(* IEC 61131-3 sources: OMJSON/, 3 files *)

(* ---- OMJSON.typ ---- *)
(********************************************************************
 * COPYRIGHT --
 ********************************************************************
 * Library: OMJSON
 * File: OMJSON.typ
 * Author: davidblackburn
 * Created: September 22, 2014
 ********************************************************************
 * Data types of library OMJSON
 ********************************************************************)

TYPE
	JSON_WS_OPCODE_enum :
		(
		JSON_WS_OPCODE_CONTINUATION := 0, (*Not supported*)
		JSON_WS_OPCODE_TEXT := 1,
		JSON_WS_OPCODE_BINARY := 2, (*Not supported*)
		JSON_WS_OPCODE_CLOSE := 8,
		JSON_WS_OPCODE_PING := 9, (*Not supported*)
		JSON_WS_OPCODE_PONG := 10 (*Not supported*)
		);
	JSON_ERR_enum :
		(
		JSON_ERR_INVALIDINPUT := 50000,
		JSON_ERR_MEMALLOC,
		JSON_ERR_MAXLEVELREACHED,
		JSON_ERR_PARSE,
		JSON_ERR_HUH,
		JSON_ERR_CACHEFULLITEMS,
		JSON_ERR_CACHEFULLVARS,
		JSON_ERR_CACHEEMPTY,
		JSON_ERR_MAXITERATIONS,
		JSON_ERR_WS_KEYNOTFOUND,
		JSON_ERR_WS_FRAGMENT,
		JSON_ERR_WS_RSV,
		JSON_ERR_WS_OPCODE,
		JSON_ERR_WS_MASK,
		JSON_ERR_WS_PAYLOADLENGTH,
		JSON_ERR_TCP_FRAGMENT,
		JSON_ERR_TCP_BAD_PACKET,
		JSON_ERR_NO_LICENSE,
		JSON_ERR_WS_MAX_CLIENTS,
		JSON_ERR_WS_INVALID_MAX_CLIENTS,
		JSON_ERR_WS_,
		JSON_ERR_
		);
	jsonWSS_client_info_typ : 	STRUCT
		Connected : BOOL;
		TimeSinceLastRequest_ms : UDINT;
		ClientIP : STRING[TCPCOMM_STRLEN_IPADDRESS];
		ClientPort : UINT;
	END_STRUCT;
	jsonWSS_client_debug_typ : 	STRUCT
		socketConnectCount : DINT;
		websocketConnectCount : DINT;
		socketDisconnectCountTimeout : DINT;
		socketDisconnectCountOpcode : DINT;
		socketDisconnectCountError : DINT;
		socketDisconnectCountRecvLength0 : DINT;
		socketInvalidCountError : DINT;
		noDataCount : DINT;
		dataCount : DINT;
		justRightCount : DINT;
		tooBigCount : DINT;
		tooSmallCount : DINT;
		doubleDataCount : DINT;
		oldDataReceived : BOOL;
	END_STRUCT;
	jsonWSServer_int_client_typ : 	STRUCT
		tcpStream : TCPStream_typ;
		pReceiveData : UDINT;
		pSendData : UDINT;
		messageBuffer : datbufBuffer_typ;
		wsConnect : jsonWSConnect;
		wsConnected : BOOL;
		wsDecode : jsonWSDecode;
		wsEncode : jsonWSEncode;
		writeVariable : jsonWriteVariable;
		readVariableList : jsonReadVariableList;
		debug : jsonWSS_client_debug_typ;
		excessDataLength : DINT;
		requestTimer : TON_10ms;
		pCache : REFERENCE TO jsonCache_typ;
	END_STRUCT;
	jsonWSServer_Internal_typ : 	STRUCT
		initialized : BOOL;
		tcpServer : TCPConnectionMgr_typ;
		client : ARRAY[0..JSON_MAI_CLIENTS]OF jsonWSServer_int_client_typ;
		requestTimer : TON_10ms;
		iClient : UINT;
		connectedClients : UINT;
		maxClients : UINT;
	END_STRUCT;
	jsonHTTPServer_Int_Debug_typ : 	STRUCT
		readSendCommand : BOOL;
	END_STRUCT;
	jsonHTTPServer_Int_Write_typ : 	STRUCT
		webService : httpService;
		pUri : UDINT;
		pRequestData : UDINT;
		ResponseHeader : httpResponseHeader_t;
		processed : BOOL;
		writeVariable : jsonWriteVariable;
	END_STRUCT;
	jsonHTTPServer_Int_Read_typ : 	STRUCT
		webService : httpService;
		pUri : UDINT;
		pRequestData : UDINT;
		ResponseHeader : httpResponseHeader_t;
		processed : BOOL;
		readVariableList : jsonReadVariableList;
	END_STRUCT;
	jsonHTTPServer_Internal_typ : 	STRUCT
		initialized : BOOL;
		read : jsonHTTPServer_Int_Read_typ;
		write : jsonHTTPServer_Int_Write_typ;
		debug : jsonHTTPServer_Int_Debug_typ;
	END_STRUCT;
	jsonWSConnect_Internal_typ : 	STRUCT
		encodeBase64 : httpEncodeBase64;
	END_STRUCT;
	JSON_TYPE_enum :
		(
		JSON_TYPE_INVALID := 0,
		JSON_TYPE_OBJECT_ELEMENT,
		JSON_TYPE_ARRAY_ELEMENT
		);
	jsonStructLevel_typ : 	STRUCT
		variable : varVariable_typ;
		iItem : UINT;
		jsonType : JSON_TYPE_enum;
	END_STRUCT;
	jsonWriteVariable_Int_typ : 	STRUCT
		initialized : BOOL;
		pJSONObject : UDINT;
		pChar : UDINT;
		iStructLevel : INT;
		structLevel : ARRAY[0..JSON_MAI_STRUCTLEVEL]OF jsonStructLevel_typ;
	END_STRUCT;
	jsonReadVariableList_Int_typ : 	STRUCT
		initialized : BOOL;
		outputBuffer : datbufBuffer_typ;
		readVariable : jsonReadVariable;
	END_STRUCT;
	jsonReadVariable_Int_typ : 	STRUCT
		initialized : BOOL;
		outputBuffer : datbufBuffer_typ;
		variableName : STRING[VAR_STRLEN_NAME];
		addVariableToCache : jsonAddVariableToCache;
	END_STRUCT;
	jsonAddVariableToCache_Int_typ : 	STRUCT
		initialized : BOOL;
		iStructLevel : INT;
		structLevel : ARRAY[0..JSON_MAI_STRUCTLEVEL]OF jsonStructLevel_typ;
	END_STRUCT;
	jsonCache_typ : 	STRUCT
		iVariable : UINT;
		variable : ARRAY[0..JSON_MAI_CACHEVAR]OF jsonCacheVariable_typ;
		iItem : UINT;
		item : ARRAY[0..JSON_MAI_CACHEITEM]OF jsonCacheItem_typ;
	END_STRUCT;
	jsonCacheVariable_typ : 	STRUCT
		name : STRING[VAR_STRLEN_NAME];
		iStart : UINT;
		iEnd : UINT;
	END_STRUCT;
	jsonCacheItem_typ : 	STRUCT
		prefix : STRING[JSON_STRLEN_PREFIX];
		variable : varVariable_typ;
		suffix : STRING[JSON_STRLEN_SUFFIX];
	END_STRUCT;
	jsonReadVarNoCache_Int_typ : 	STRUCT
		initialized : BOOL;
		outputBuffer : datbufBuffer_typ;
		iStructLevel : INT;
		structLevel : ARRAY[0..JSON_MAI_STRUCTLEVEL]OF jsonStructLevel_typ;
	END_STRUCT;
END_TYPE

(* ---- OMJSON.fun ---- *)
(********************************************************************
 * COPYRIGHT --
 ********************************************************************
 * Library: OMJSON
 * File: OMJSON.fun
 * Author: davidblackburn
 * Created: September 22, 2014
 ********************************************************************
 * Functions and function blocks of library OMJSON
 ********************************************************************)

FUNCTION_BLOCK jsonWebSocketServer (*Serve variables via JSON and WebSockets*) (*$GROUP=User*)
	VAR_INPUT
		pCacheArray : UDINT; (*Address of the variable cache array. Number of elements in array needs to be equal to numClients*)
		maxClients : UINT; (*Number of clients supported at a time. 0 defaults to 1*)
		ServerIP : STRING[TCPCOMM_STRLEN_IPADDRESS]; (*IP Address of the server*)
		ServerPort : UINT; (*Port to be used by server*)
		BufferSize : UDINT; (*Size of buffers. N buffers will be allocated, so the total memory requirement is N*BufferSize.*)
		MaxIterations : UDINT; (*Maximum number of iterations for looping through variables.*)
		AcknowledgeError : BOOL; (*Acknowledge errors. Automatically reset by FUB.*)
		Timeout : UDINT; (*Max time in miliseconds since last message from client before forcing disconnect*)
	END_VAR
	VAR_OUTPUT
		ClientInfo : ARRAY[0..JSON_MAI_CLIENTS] OF jsonWSS_client_info_typ;
		Error : BOOL;
		ErrorID : UINT;
		ErrorString : STRING[JSON_STRLEN_ERROR];
	END_VAR
	VAR
		internal : jsonWSServer_Internal_typ;
	END_VAR
END_FUNCTION_BLOCK

FUNCTION_BLOCK jsonWSConnect (*Negotiate a new WebSocket connection*) (*$GROUP=User,$CAT=User,$GROUPICON=User.png,$CATICON=User.png*)
	VAR_INPUT
		pInputMessage : UDINT;
		pOutputMessage : UDINT;
		MaxOutputMessageLength : UDINT;
	END_VAR
	VAR_OUTPUT
		Status : UINT;
		OutputMessageLength : UDINT;
	END_VAR
	VAR
		internal : jsonWSConnect_Internal_typ;
	END_VAR
END_FUNCTION_BLOCK

FUNCTION_BLOCK jsonWSDecode (*Decode a WebSocket frame*) (*$GROUP=User,$CAT=User,$GROUPICON=User.png,$CATICON=User.png*)
	VAR_INPUT
		pFrame : UDINT;
	END_VAR
	VAR_OUTPUT
		Status : UINT;
		FIN : BOOL;
		RSV : USINT;
		OpCode : USINT;
		MASK : BOOL;
		MaskingKey : ARRAY[0..3] OF USINT;
		pPayloadData : UDINT;
		HeaderLength : UDINT;
		PayloadLength : UDINT;
		FrameLength : UDINT;
	END_VAR
END_FUNCTION_BLOCK

FUNCTION_BLOCK jsonWSEncode (*Encode data into a WebSocket frame*) (*$GROUP=User,$CAT=User,$GROUPICON=User.png,$CATICON=User.png*)
	VAR_INPUT
		pFrame : UDINT;
		MaxFrameLength : UDINT;
		FIN : BOOL;
		RSV : USINT;
		OpCode : USINT;
		MASK : BOOL; (*NOT SUPPORTED*)
		PayloadLength : UDINT;
		MaskingKey : ARRAY[0..3] OF USINT; (*NOT SUPPORTED*)
		pPayloadData : UDINT;
	END_VAR
	VAR_OUTPUT
		Status : UINT;
		FrameLength : UDINT;
	END_VAR
END_FUNCTION_BLOCK

FUNCTION_BLOCK jsonHTTPServer (*Serve variables via JSON and HTTP*) (*$GROUP=User*)
	VAR_INPUT
		pCache : UDINT; (*Address of the variable cache*)
		ServiceNamePrefix : STRING[JSON_STRLEN_SERVICENAMEPREFIX]; (*Optional service name prefix*)
		BufferSize : UDINT; (*Size of buffers. N buffers will be allocated, so the total memory requirement is N*BufferSize.*)
		MaxIterations : UDINT; (*Maximum number of iterations for looping through variables.*)
		AcknowledgeError : BOOL; (*Acknowledge errors. Automatically reset by FUB.*)
	END_VAR
	VAR_OUTPUT
		Error : BOOL;
		ErrorID : UINT;
		ErrorString : STRING[JSON_STRLEN_ERROR];
	END_VAR
	VAR
		internal : jsonHTTPServer_Internal_typ;
	END_VAR
END_FUNCTION_BLOCK

FUNCTION_BLOCK jsonWriteVariable (*Write variable values received as a JSON object*) (*$GROUP=User*)
	VAR_INPUT
		pJSONObject : UDINT; (*Address of the JSON object*)
		MaxJSONObjectLength : UDINT; (*Maximum length of the JSON object*)
		MaxIterations : UDINT; (*Maximum number of iterations for expanding structures*)
	END_VAR
	VAR_OUTPUT
		Status : UINT; (*0 = Done, 65535 = Busy, other values are errors*)
	END_VAR
	VAR
		internal : jsonWriteVariable_Int_typ;
	END_VAR
END_FUNCTION_BLOCK

FUNCTION_BLOCK jsonReadVariableList (*Convert a list of variables into a JSON object*) (*$GROUP=User*)
	VAR_INPUT
		pVariableList : UDINT;
		pCache : UDINT;
		BufferSize : UDINT;
		MaxIterations : UDINT;
	END_VAR
	VAR_OUTPUT
		Status : UINT;
		pJSONObject : UDINT;
		JSONObjectLength : UDINT;
	END_VAR
	VAR
		internal : jsonReadVariableList_Int_typ;
	END_VAR
END_FUNCTION_BLOCK

FUNCTION_BLOCK jsonReadVariable (*Convert a variable into a JSON object*) (*$GROUP=User*)
	VAR_INPUT
		pVariableName : UDINT;
		pCache : UDINT;
		BufferSize : UDINT;
		MaxIterations : UDINT;
	END_VAR
	VAR_OUTPUT
		Status : UINT;
		pJSONObject : UDINT;
		JSONObjectLength : UDINT;
	END_VAR
	VAR
		internal : jsonReadVariable_Int_typ;
	END_VAR
END_FUNCTION_BLOCK

FUNCTION_BLOCK jsonAddVariableToCache (*Add a variable to the JSON variable cache*) (*$GROUP=User*)
	VAR_INPUT
		pVariableName : UDINT;
		pCache : UDINT;
		MaxIterations : UDINT;
	END_VAR
	VAR_OUTPUT
		Status : UINT;
		iVariable : UINT;
	END_VAR
	VAR
		internal : jsonAddVariableToCache_Int_typ;
	END_VAR
END_FUNCTION_BLOCK

FUNCTION_BLOCK jsonReadVariableNoCache (*Convert a variable into a JSON object without caching*) (*$GROUP=User*)
	VAR_INPUT
		pVariableName : UDINT; (*Address of name of variable to convert to JSON*)
		BufferSize : UDINT; (*Size of internal data buffer*)
		MaxIterations : UDINT; (*Maximum number of iterations for expanding structures*)
	END_VAR
	VAR_OUTPUT
		Status : UINT; (*0 = Done, 65535 = Busy, other values are errors*)
		pJSONObject : UDINT; (*Address of the generated JSON object*)
		JSONObjectLength : UDINT; (*Length of the generated JSON object*)
	END_VAR
	VAR
		internal : jsonReadVarNoCache_Int_typ;
	END_VAR
END_FUNCTION_BLOCK

FUNCTION jsonUnescape : UDINT (*Unescape JSON string*)
	VAR_INPUT
		pDest : UDINT;
		pSrc : UDINT;
		maxLength : UDINT;
		reentry : UDINT;
	END_VAR
END_FUNCTION

FUNCTION jsonEscape : UDINT (*Escape JSON string*)
	VAR_INPUT
		pDest : UDINT;
		pSrc : UDINT;
		maxLength : UDINT;
		reentry : UDINT;
	END_VAR
END_FUNCTION

(* ---- OMJSON.var ---- *)
(********************************************************************
 * COPYRIGHT --
 ********************************************************************
 * Library: OMJSON
 * File: OMJSON.var
 * Author: davidblackburn
 * Created: September 22, 2014
 ********************************************************************
 * Constants of library OMJSON
 ********************************************************************)
VAR CONSTANT
	JSON_DEFAULT_SERVERPORT : UINT := 8000;
	JSON_DEFAULT_BUFFERSIZE : UDINT := 100000;
	JSON_DEFAULT_MAXJSONOBJECTLENGTH : UDINT := 100000;
	JSON_DEFAULT_MAXITERATIONS : UDINT := 10000;
	JSON_DEFAULT_TIMEOUT : UDINT := 30000;
	JSON_MAX_CLIENTS : UINT := 5;
	JSON_MAI_CLIENTS : UINT := JSON_MAX_CLIENTS-1;
	JSON_MAI_STRUCTLEVEL : USINT := 19;
	JSON_MAI_CACHEVAR : UINT := 400;
	JSON_MAI_CACHEITEM : UINT := 20000;
	JSON_STRLEN_ERROR : UINT := 320;
	JSON_STRLEN_PREFIX : UINT := 400;
	JSON_STRLEN_SUFFIX : UINT := 20;
	JSON_STRLEN_IP : UINT := 15;
	JSON_STRLEN_SERVICENAMEPREFIX : UINT := 20;
	JSON_STRLEN_WSKEYHEADER : UINT := 18;
	JSON_STRLEN_WSCONNECTMESSAGE : UINT := 129;
	JSON_WS_MAGICSTRING : STRING[36] := '258EAFA5-E914-47DA-95CA-C5AB0DC85B11';
END_VAR
